FUNCTION_BLOCK FB_NoLimitSwitch IMPLEMENTS I_LimitSwitch
VAR_INPUT
END_VAR
VAR_OUTPUT
END_VAR
VAR
END_VAR

END_FUNCTION_BLOCK

(* stored: Version 1.1.0.1
   POU FB_NoLimitSwitch: Id {71d6e03f-8fca-46aa-9c3d-cbcac4ee8f67}, SpecialFunc None *)
